FUNCTION Convert_DINT_TO_DWORD : Hresult
VAR_INPUT
	in : DINT;
	out : REFERENCE TO DWORD;
END_VAR
VAR
	converted : DWORD;
END_VAR
VAR CONSTANT
	INCOMPATIBLE : HRESULT := 16#9811070E;
END_VAR

converted := DINT_TO_DWORD(in);

IF (DWORD_TO_DINT(converted) <> in) THEN
	Convert_DINT_TO_DWORD := INCOMPATIBLE;
	RETURN;
END_IF

out := converted;

END_FUNCTION

(* stored: Version 1.1.0.1, ProductVersion 3.1.4024.12
   POU Convert_DINT_TO_DWORD: Id {922dedef-ed7f-426a-a829-2b5ff1a57361}, SpecialFunc None *)
